{attribute 'GeneratedUsingTerminal: EL3773-0000-0016'}
{attribute addProperty BoxType "EL3773-0000-0016"}
{attribute addProperty Id "I1_SAMPLESAT %I*I1_SAMPLES_2D13B74B20"}
{attribute addProperty CRC "839495983"}
{attribute addProperty Size "20"}
TYPE L1_Current_Samples_3209B12F EXTENDS InputBase_8311D824 :
STRUCT
	{attribute addProperty Name "I1_SAMPLES"}
	I1_SAMPLES AT %I* : I1_SAMPLES_2D13B74B;
END_STRUCT
END_TYPE

(* stored: Version 1.2.0.0, ProductVersion 3.1.4024.9
   DUT L1_Current_Samples_3209B12F: Id {0c44e3dc-73b7-4ed5-b79f-34a31427e41f} *)
